FUNCTION IIRFilter : REAL
VAR_INPUT
	newValue : REAL;
	filterStrength : REAL;
END_VAR
VAR_IN_OUT
	value : REAL;
END_VAR
VAR
END_VAR

value := newValue*(1-filterStrength) + value*filterStrength;

END_FUNCTION

(* stored: Version 1.1.0.1, ProductVersion 3.1.4024.9
   POU IIRFilter: Id {b7b3d10b-2037-4039-9c3c-7bae6cb0d870}, SpecialFunc None *)
